{attribute 'GeneratedUsingTerminal: AT2050-0500-0017'}
{attribute addProperty BoxType "AT2050-0500-0017"}
{attribute addProperty Id "A_0096_AT2025_5250_0017_AT2025_5250AT2025_33A3DF1B80"}
{attribute addProperty CRC "1066893127"}
{attribute addProperty Size "80"}
TYPE A_0048_AT2050_0500_0017_3F977F47 EXTENDS AT2050_2EA6C9BF :
STRUCT
	{attribute addProperty Name "A_0096_AT2025_5250_0017_AT2025_5250"}
	{attribute addProperty PreviousPort "A_0048(AT2050-0500-0017) : B"}
	A_0096_AT2025_5250_0017_AT2025_5250 : AT2025_33A3DF1B;
END_STRUCT
END_TYPE

(* stored: Version 1.2.0.0, ProductVersion 3.1.4024.9
   DUT A_0048_AT2050_0500_0017_3F977F47: Id {868d5d02-7756-4a97-a08b-dc68a6ba2b05} *)
